PROGRAM Permissives
VAR
	
	
END_VAR

//charge relay 
IF (MCP_IO.MagDriver[1].ChargeRelayClose = TRUE AND 
	MCP_IO.MagDriver[2].ChargeRelayClose = TRUE AND
	MCP_IO.MagDriver[3].ChargeRelayClose = TRUE AND 
	MCP_IO.MagDriver[4].ChargeRelayClose = TRUE AND 
	MCP_IO.MagDriver[5].ChargeRelayClose = TRUE AND 
	MCP_IO.MagDriver[6].ChargeRelayClose = TRUE) OR HMI_DB.AllChargeRelayCloseBP = TRUE
	THEN 
		Permissives_DB.AllChargeRelayClosed := TRUE;
	ELSIF 
		MCP_IO.MagDriver[1].ChargeRelayClose = FALSE AND 
		MCP_IO.MagDriver[2].ChargeRelayClose = FALSE AND
		MCP_IO.MagDriver[3].ChargeRelayClose = FALSE AND 
		MCP_IO.MagDriver[4].ChargeRelayClose = FALSE AND 
		MCP_IO.MagDriver[5].ChargeRelayClose = FALSE AND 
		MCP_IO.MagDriver[6].ChargeRelayClose = FALSE
	THEN
		Permissives_DB.AllChargeRelayClosed := FALSE;
END_IF;

//dump relay
IF (MCP_IO.MagDriver[1].DumpRelayOpen = TRUE AND 
	MCP_IO.MagDriver[2].DumpRelayOpen = TRUE AND
	MCP_IO.MagDriver[3].DumpRelayOpen = TRUE AND
	
	MCP_IO.MagDriver[4].DumpRelayOpen = TRUE AND 
	MCP_IO.MagDriver[5].DumpRelayOpen = TRUE AND
	MCP_IO.MagDriver[6].DumpRelayOpen = TRUE) OR HMI_DB.AllDumpRelaysOpenBP = TRUE
	THEN
		Permissives_DB.AllDumpRelayOpen := TRUE;
		ELSIF
			MCP_IO.MagDriver[1].DumpRelayOpen = FALSE AND 
			MCP_IO.MagDriver[2].DumpRelayOpen = FALSE AND
			MCP_IO.MagDriver[3].DumpRelayOpen = FALSE AND
			MCP_IO.MagDriver[4].DumpRelayOpen = FALSE AND
			MCP_IO.MagDriver[5].DumpRelayOpen = FALSE AND
			MCP_IO.MagDriver[6].DumpRelayOpen = FALSE 
		THEN
			Permissives_DB.AllDumpRelayOpen := FALSE;
END_IF;

IF Permissives_DB.AllChargeRelayClosed = TRUE AND 
	Permissives_DB.AllDumpRelayOpen = TRUE  AND 
	Permissives_DB.AllDumpResTempOK = TRUE //voltmonitor board has missing packets, so this might be sensitive and might need to bypass	
	THEN
		Permissives_DB.ReadyToCharge := TRUE;
	ELSE 
		Permissives_DB.ReadyToCharge := FALSE;
END_IF

//charger dc ok
IF MCP_IO.Charger[1].DCOK = TRUE AND 
	MCP_IO.Charger[2].DCOK = TRUE AND 
	MCP_IO.Charger[3].DCOK = TRUE AND
	MCP_IO.Charger[4].DCOK = TRUE AND
	MCP_IO.Charger[5].DCOK = TRUE AND
	MCP_IO.Charger[6].DCOK = TRUE 
	THEN
		Permissives_DB.AllChargerDCOK := TRUE;
	ELSE 
		Permissives_DB.AllChargerDCOK := FALSE;
END_IF
//charger ac ok
IF MCP_IO.Charger[1].ACOK = TRUE AND 
	MCP_IO.Charger[2].ACOK = TRUE AND 
	MCP_IO.Charger[3].ACOK = TRUE AND
	MCP_IO.Charger[4].ACOK = TRUE AND
	MCP_IO.Charger[5].ACOK = TRUE AND
	MCP_IO.Charger[6].ACOK = TRUE 
	THEN
		Permissives_DB.AllChargerACOK := TRUE;
	ELSE 
		Permissives_DB.AllChargerACOK := FALSE;
END_IF

// temperature 
IF MCP_IO.Charger[1].OverTemp = FALSE AND 
	MCP_IO.Charger[2].OverTemp = FALSE AND 
	MCP_IO.Charger[3].OverTemp = FALSE AND
	MCP_IO.Charger[4].OverTemp = FALSE AND
	MCP_IO.Charger[5].OverTemp = FALSE AND
	MCP_IO.Charger[6].OverTemp = FALSE 
	THEN
		Permissives_DB.AllChargerTempOK := TRUE;
	ELSE 
		Permissives_DB.AllChargerTempOK := FALSE;
END_IF

//dump resistor temp 
Permissives_DB.TempThres := HMI_DB.DumpResTempThres;

IF (MCP_IO.MagDriver[1].DumpResistorTemp < Permissives_DB.TempThres AND
	MCP_IO.MagDriver[2].DumpResistorTemp < Permissives_DB.TempThres AND
	MCP_IO.MagDriver[3].DumpResistorTemp < Permissives_DB.TempThres AND
	MCP_IO.MagDriver[4].DumpResistorTemp < Permissives_DB.TempThres AND
	MCP_IO.MagDriver[5].DumpResistorTemp < Permissives_DB.TempThres AND
	MCP_IO.MagDriver[6].DumpResistorTemp < Permissives_DB.TempThres) OR HMI_DB.AllDumpRTempOKBP = TRUE
	THEN 
		Permissives_DB.AllDumpResTempOK := TRUE;
		ELSE
			Permissives_DB.AllDumpResTempOK := FALSE;
END_IF

//cap voltage
IF (MCP_IO.MagDriver[1].Cap[1].CapVoltage <= Permissives_DB.CapVoltageThres AND
	MCP_IO.MagDriver[1].Cap[2].CapVoltage <= Permissives_DB.CapVoltageThres AND
	MCP_IO.MagDriver[2].Cap[1].CapVoltage <= Permissives_DB.CapVoltageThres AND
	MCP_IO.MagDriver[2].Cap[2].CapVoltage <= Permissives_DB.CapVoltageThres AND
	MCP_IO.MagDriver[3].Cap[1].CapVoltage <= Permissives_DB.CapVoltageThres AND
	MCP_IO.MagDriver[3].Cap[2].CapVoltage <= Permissives_DB.CapVoltageThres AND
	MCP_IO.MagDriver[4].Cap[1].CapVoltage <= Permissives_DB.CapVoltageThres AND
	MCP_IO.MagDriver[4].Cap[2].CapVoltage <= Permissives_DB.CapVoltageThres AND
	MCP_IO.MagDriver[5].Cap[1].CapVoltage <= Permissives_DB.CapVoltageThres AND
	MCP_IO.MagDriver[5].Cap[2].CapVoltage <= Permissives_DB.CapVoltageThres AND
	MCP_IO.MagDriver[6].Cap[1].CapVoltage <= Permissives_DB.CapVoltageThres AND
	MCP_IO.MagDriver[6].Cap[2].CapVoltage <= Permissives_DB.CapVoltageThres) OR HMI_DB.AllCapsDischargedBP = TRUE 
(*  AND all other module voltage feedback <= 40, might need the -ve end & check for valid data*) 
	THEN
		Permissives_DB.AllCapsDischarged := TRUE;
	ELSE 
		Permissives_DB.AllCapsDischarged := FALSE;
END_IF

IF MCP_IO.MagDriver[1].SCR_ready_to_fire AND 
	MCP_IO.MagDriver[2].SCR_ready_to_fire AND 
	MCP_IO.MagDriver[3].SCR_ready_to_fire AND 
	MCP_IO.MagDriver[4].SCR_ready_to_fire AND 
	MCP_IO.MagDriver[5].SCR_ready_to_fire AND 
	MCP_IO.MagDriver[6].SCR_ready_to_fire 
	THEN 
		Permissives_DB.AllSCRreadyToFire := TRUE;
		ELSE
			Permissives_DB.AllSCRreadyToFire := FALSE;
END_IF;

IF (//Permissives_DB.AllChargerInhibitON	= TRUE AND 
	Permissives_DB.AllDumpRelayOpen = FALSE AND 
	Permissives_DB.AllCapsDischarged = TRUE) OR HMI_DB.SystemSafeBP = TRUE 
THEN
	(*MCP_IO.Charger[2].voltageFeedback <= 10 AND *)
	Permissives_DB.SystemIsSafe := TRUE;
	ELSE
		Permissives_DB.SystemIsSafe := FALSE;
END_IF
		
IF Permissives_DB.AllCapsDischarged = TRUE THEN 
	MCP_IO.TurnONSystemChargedLED := FALSE; //for status light only
END_IF

//MCP_IO.Charger[i].ACOK , DCOK, TEMPOK...

// might or might not beused for the seq
IF MCP_IO.PSU1_DCOK = TRUE AND MCP_IO.Charger[1].ACOK = TRUE  THEN
	Trips_DB.AllDCpsuOK := TRUE;
	ELSE
		Trips_DB.AllDCpsuOK := FALSE;
END_IF

IF MCP_IO.MasterStopPB_NotPressed = FALSE THEN 
	Trips_DB.MasterSTOPPressed := TRUE;
	ELSE
		Trips_DB.MasterSTOPPressed := FALSE;
END_IF

//add logic for e stop
IF MCP_IO.CageEstopCircuitOK = FALSE OR Trips_DB.AnyEstopPressed = FALSE THEN 
	Trips_DB.AnyEstopPressed := TRUE;
END_IF

END_PROGRAM

(* stored: Version 1.1.0.1, ProductVersion 3.1.4024.11
   POU Permissives: Id {639d0291-603e-4994-93d7-3ec14345fa0c}, SpecialFunc None *)
